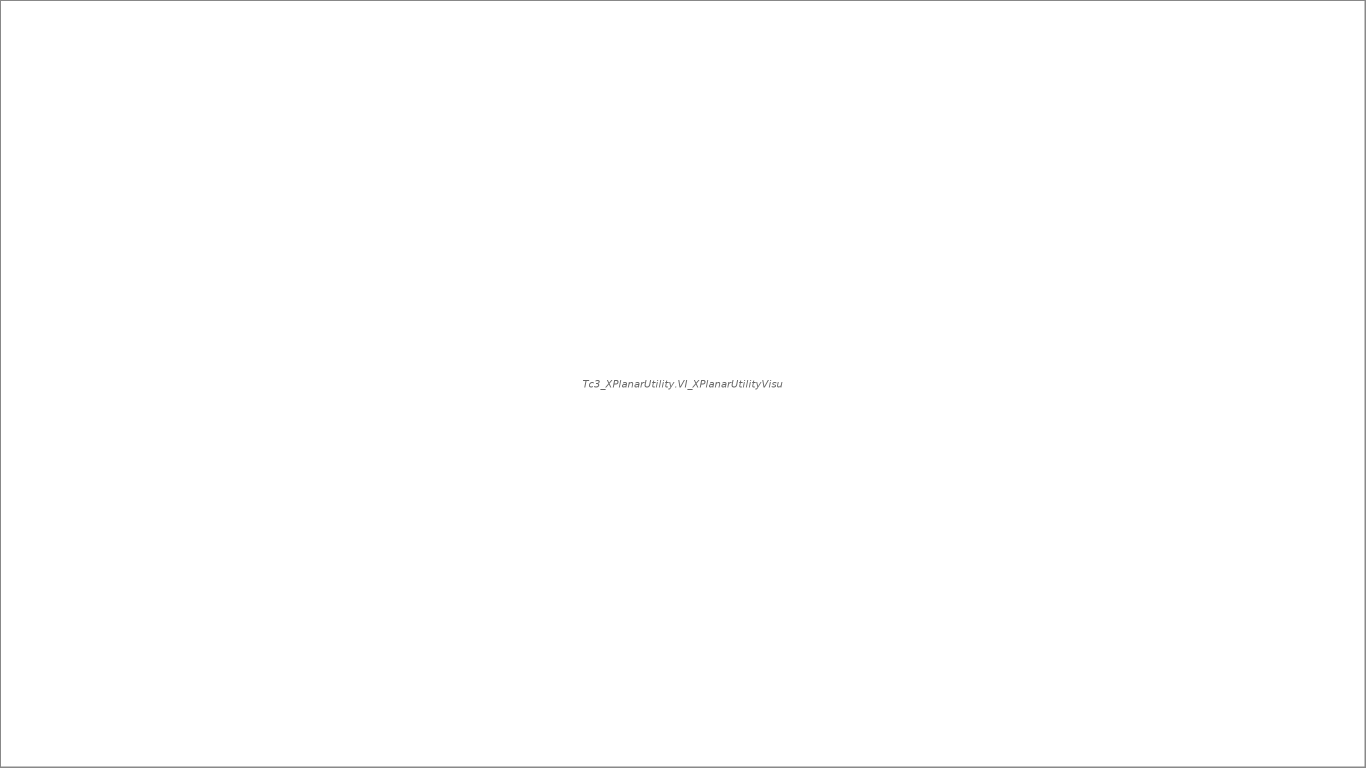
VISUALIZATION Visu_XPlanarUtility  // 1366x768
    Frame (0,0 1366x768)
        shows Tc3_XPlanarUtility.VI_XPlanarUtilityVisu()
END_VISUALIZATION

(* stored: Version 1.1.0.1, ProductVersion 3.1.4024.9
   Visu Visu_XPlanarUtility: Id {c8f38fc5-bf21-43eb-8773-c5d5fcd0e3e4} *)
